Omron Sysmac Studio project ewon_1 (Sysmac Studio 1.23.0.14, StandardProject)

# Controller new_Controller_0: NX1P2-1040DT1 version 1.18
Task PrimaryTask (priority 4, period or condition 2000): Programa0

VAR_GLOBAL
    motor : BOOL;  (* at BuiltInIO://cpu/#0/Output_Bit_00 *)
END_VAR
VAR_GLOBAL RETAIN
    marcha AT %D800.0 : BOOL;  (* published *)
    paro AT %D800.1 : BOOL;  (* published *)
    marca_motor AT %D800.2 : BOOL;  (* published *)
    tiempo_encendido AT %D801 : INT;  (* published *)
    temporizar_encendido AT %D805.0 : BOOL;  (* published *)
    tiempo_pasado AT %D806 : INT;  (* published *)
END_VAR

PROGRAM Programa0
VAR
    retardo_desconexion : TOF;
    encendido_temporizado : TON;
    timerDat : _sTimer;
    timer_out : BOOL;
    PT : UINT;
    ET : UINT;
END_VAR
VAR_EXTERNAL
    marcha : BOOL;
    motor : BOOL;
    paro : BOOL;
    tiempo_encendido : INT;
    tiempo_pasado : INT;
    temporizar_encendido : BOOL;
    marca_motor : BOOL;
END_VAR
VAR
    _t1 : BOOL;
END_VAR

(* Section Sección0: ladder, written here as Structured Text *)

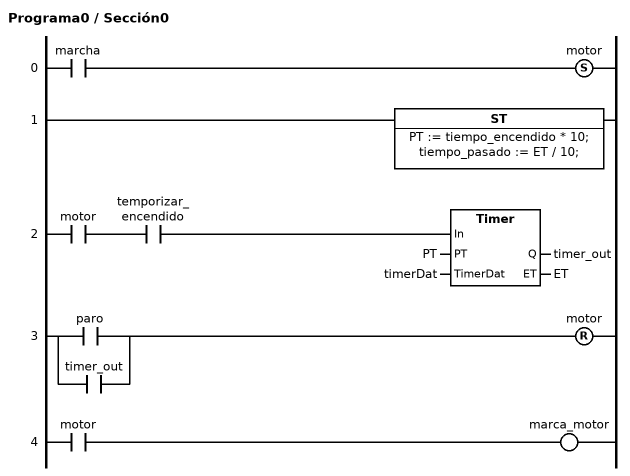
(* Rung 0 *)
IF marcha THEN motor := TRUE; END_IF;
(* Rung 1 *)
PT := tiempo_encendido * 10;
tiempo_pasado := ET / 10;
(* Rung 2 *)
_t1 := Timer(In := motor AND temporizar_encendido, PT := PT, TimerDat := timerDat, Q => timer_out, ET => ET);
(* Rung 3 *)
IF paro OR timer_out THEN motor := FALSE; END_IF;
(* Rung 4 *)
marca_motor := motor;
END_PROGRAM